// SIMATIC S7-200 project (STEP 7-Micro/WIN), CPU 224 AM REL 21.02

ORGANIZATION_BLOCK 主程序:OB1
TITLE=程序注释
BEGIN
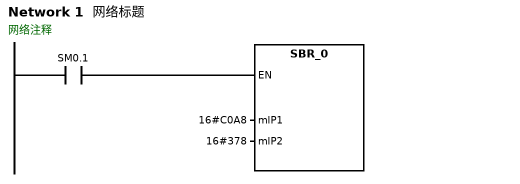
Network 1 // 网络标题
// 网络注释
LD     SM0.1
CALL   SBR_0:SBR0, 16#C0A8, 16#378
END_ORGANIZATION_BLOCK

SUBROUTINE_BLOCK SBR_0:SBR0
TITLE=子程序注释
VAR_INPUT
mlP1:WORD;	// LW0 
mlP2:WORD;	// LW2 
END_VAR
BEGIN
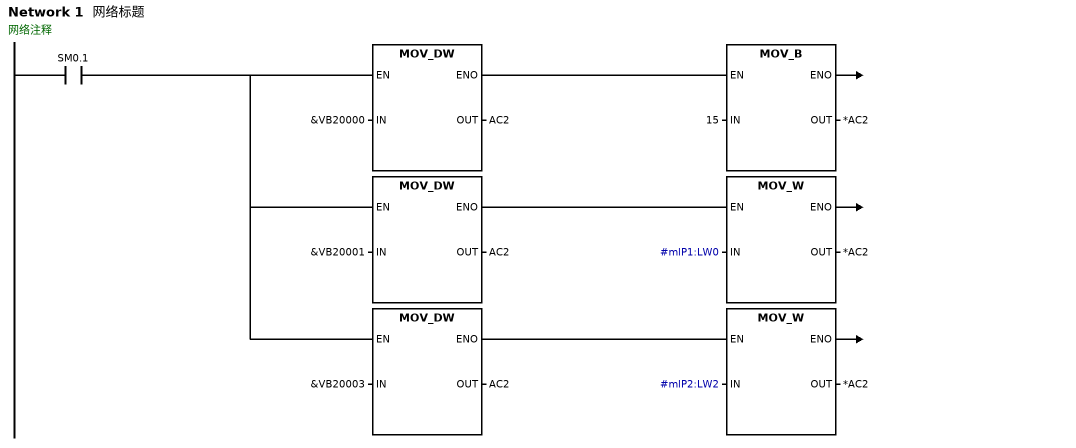
Network 1 // 网络标题
// 网络注释
// (network saved uncompiled; LAD cells follow)
// row 0: c0 -| |- SM0.1  c1 -- v  c2 --  c3 [MOV_DW EN:=power@row0, IN:=&VB20000, ENO=>power, OUT=>AC2]  c4 --  c5 --  c6 [MOV_B EN:=power@row0, IN:=15, ENO=>power, OUT=>*AC2]  c7 ->
// row 1: c1 ^v  c3 [box]  c6 [box]
// row 2: c1 ^v  c2 --  c3 [MOV_DW EN:=power@row2, IN:=&VB20001, ENO=>power, OUT=>AC2]  c4 --  c5 --  c6 [MOV_W EN:=power@row2, IN:=#mlP1:LW0, ENO=>power, OUT=>*AC2]  c7 ->
// row 3: c1 ^v  c3 [box]  c6 [box]
// row 4: c1 ^  c2 --  c3 [MOV_DW EN:=power@row4, IN:=&VB20003, ENO=>power, OUT=>AC2]  c4 --  c5 --  c6 [MOV_W EN:=power@row4, IN:=#mlP2:LW2, ENO=>power, OUT=>*AC2]  c7 ->
// row 5: c3 [box]  c6 [box]
END_SUBROUTINE_BLOCK
